// TIA Portal V20 export
// export: Created 2026-07-16T12:59:12.3306694Z, ExportSetting WithDefaults, DisplayName Totally Integrated Automation Portal, DisplayVersion V20 Update 5, DisplayName TIA Portal Openness, DisplayVersion V20 Update 4, DisplayName TIA Portal Version Control Interface, DisplayVersion V20 Update 5, DisplayName SINAMICS Startdrive Advanced, DisplayVersion V20, DisplayName SINAMICS DCC, DisplayVersion V20, DisplayName SINAMICS Startdrive G130, G150, S120, S150, SINAMICS MV, G220, S200, S210, DisplayVersion V20, DisplayName SINAMICS Startdrive G110M, G120, G120C, G120D, G120P, G115D, DisplayVersion V20, DisplayName STEP 7 Professional, DisplayVersion V20 Update 5, DisplayName STEP 7 Safety, DisplayVersion V20 Update 2, DisplayName WinCC Basic/Comfort/Advanced, DisplayVersion V20 Update 5, DisplayName WinCC Unified, DisplayVersion V20 Update 5
ORGANIZATION_BLOCK "Main"   // OB1, LAD, ProgramCycle
TITLE = "Main Program Sweep (Cycle)"
{ S7_Optimized_Access := 'TRUE' }
VERSION : 0.1
// stored: AutoNumber true, IsIECCheckEnabled false, SetENOAutomatically false
   VAR_INPUT
      Initial_Call : Bool;   // Initial call of this OB
      Remanence : Bool;   // =True, if remanent data are available
   END_VAR
BEGIN

REGION Network 1: Input Mapping
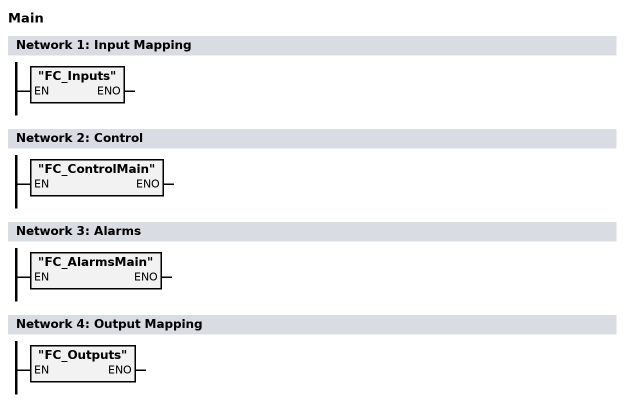
   RUNG wire#powerrail
      "FC_Inputs"()
   END_RUNG
   // the same network as SCL:
   "FC_Inputs"();
END_REGION

REGION Network 2: Control
   RUNG wire#powerrail
      "FC_ControlMain"()
   END_RUNG
   // the same network as SCL:
   "FC_ControlMain"();
END_REGION

REGION Network 3: Alarms
   RUNG wire#powerrail
      "FC_AlarmsMain"()
   END_RUNG
   // the same network as SCL:
   "FC_AlarmsMain"();
END_REGION

REGION Network 4: Output Mapping
   RUNG wire#powerrail
      "FC_Outputs"()
   END_RUNG
   // the same network as SCL:
   "FC_Outputs"();
END_REGION
END_ORGANIZATION_BLOCK
